FUNCTION_BLOCK FB_Conveyer IMPLEMENTS I_Conveyer

VAR
END_VAR

{warning 'add method implementation '}
METHOD Start : BOOL
Start := GVL_HMI.bConveyerRunning := TRUE;
END_METHOD

{warning 'add method implementation '}
METHOD Stop : BOOL
Stop := GVL_HMI.bConveyerRunning := FALSE;
END_METHOD

END_FUNCTION_BLOCK

(* stored: Version 1.1.0.1, ProductVersion 3.1.4024.16
   POU FB_Conveyer: Id {9cc60f3c-fe0a-4a51-bb77-a7cc286b637c}, SpecialFunc None
   Method Start: Id {5f11bbe9-a744-40ff-9fa2-2b141ea96d70}
   Method Stop: Id {e594c64a-6bac-48ae-aa9b-1c5ddd37c96b} *)
